// TwinCAT 3 PLC project SimpleTcUnitExampleProject
// Title: TcUnit simple example
// Company: www.tcunit.org
// Author: Jakob Sagatowski
// ProjectVersion: 1.0.0.0
// Description: This library is a demonstration of the TcUnit framework, which is a TwinCAT unit testing framework. See www.tcunit.org for more information.
// ProgramVersion: 3.1.4022.3
// libraries:
//   Tc2_Standard, * (Beckhoff Automation GmbH)
//   Tc2_System, * (Beckhoff Automation GmbH)
//   Tc3_Module, * (Beckhoff Automation GmbH)
//   TcUnit, * (www.tcunit.org)
// project tree:
//   / PlcTask.TcTTO
//   POUs/ FB_Sum.TcPOU
//   Test/ FB_Sum_Test.TcPOU, PRG_TEST.TcPOU
// real-time tasks:
//   TASK PlcTask: cycle T#10ms, priority 20, ADS port 350

CONFIGURATION SimpleTcUnitExampleProject
    RESOURCE PLC ON TwinCAT3
        TASK PlcTask(INTERVAL := T#10ms, PRIORITY := 20);
        PROGRAM PRG_TEST WITH PlcTask : PRG_TEST;
    END_RESOURCE
END_CONFIGURATION

// ---- Test/PRG_TEST.TcPOU
PROGRAM PRG_TEST
VAR
	fbSum_Test : FB_Sum_Test;
END_VAR

TcUnit.RUN();

END_PROGRAM

// ---- Test/FB_Sum_Test.TcPOU
FUNCTION_BLOCK FB_Sum_Test EXTENDS TcUnit.FB_TestSuite
VAR
END_VAR

TwoPlusTwoEqualsFour();
ZeroPlusZeroEqualsZero();

METHOD PRIVATE TwoPlusTwoEqualsFour
VAR
	Sum : FB_Sum;
	Result : UINT;
    ExpectedSum : UINT := 4;
END_VAR
TEST('TwoPlusTwoEqualsFour');

Sum(one := 2, two := 2, result => Result);

AssertEquals(Expected := ExpectedSum,
             Actual := Result,
             Message := 'The calculation is not correct');

TEST_FINISHED();
END_METHOD

METHOD PRIVATE ZeroPlusZeroEqualsZero
VAR
	Sum : FB_Sum;
	Result : UINT;
    ExpectedSum : UINT := 0;
END_VAR
TEST('ZeroPlusZeroEqualsZero');

Sum(one := 0, two := 0, result => Result);

AssertEquals(Expected := ExpectedSum,
             Actual := Result,
             Message := 'The calculation is not correct');

TEST_FINISHED();
END_METHOD

END_FUNCTION_BLOCK

// ---- POUs/FB_Sum.TcPOU
FUNCTION_BLOCK FB_Sum
VAR_INPUT
	one : UINT;
	two : UINT;
END_VAR
VAR_OUTPUT
	result : UINT;
END_VAR

result := one + two;

END_FUNCTION_BLOCK
